Staubli VAL3: initToSafePt.pgx

program initToSafePt(string x_sName)
  local num i
  local num j
  local num l_n
begin
  l_n=-9999
  for i=0 to size(sml:box[x_sName].pPointRx)-1
    if sml:box[x_sName].pPointRx[i].trsf.z>l_n and left(sml:box[x_sName].comment[i],1)=="#"
      j=i
    endIf
  endFor
  sml:box[x_sName].pToSafePt=sml:box[x_sName].pPointRx[j]
end
